FUNCTION_BLOCK FINAL TcoContextNfCompatibility EXTENDS TcoContextCompatibility
VAR
END_VAR

METHOD PROTECTED FINAL Main
END_METHOD

METHOD PUBLIC VolatileClose
THIS^._Close();
END_METHOD

METHOD PUBLIC VolatileOpen
THIS^._Open();
END_METHOD

END_FUNCTION_BLOCK

(* stored: Version 1.1.0.1, ProductVersion 3.1.4024.6
   POU TcoContextNfCompatibility: Id {ecb51e5b-aa76-4bdc-9a90-de522a9d69ee}, SpecialFunc None
   Method Main: Id {cc2e5ac9-9371-4d57-a8ee-2f167ab4c0c4}
   Method VolatileClose: Id {99ea6149-a9cb-4e95-8e93-dc1156107c90}
   Method VolatileOpen: Id {15ea9abe-e110-469a-b218-80cc9ec12892} *)
